{attribute addProperty BoxType "BK1120-0000-0000"}
{attribute addProperty Id "Term_374_KL1002KL1002_D229A9CA00"}
{attribute addProperty CRC "2703046566"}
{attribute addProperty SizeInBites "0"}
{attribute addProperty SizeInBytes "0"}
TYPE A_0001_BK1120_0000_0000_A11D37A6 EXTENDS BK1120_D3F02A0D :
STRUCT
	{attribute addProperty Name "Term_374_KL1002"}
	Term_374_KL1002 : KL1002_D229A9CA;
END_STRUCT
END_TYPE

(* stored: Version 1.2.0.0, ProductVersion 3.1.4024.9
   DUT A_0001_BK1120_0000_0000_A11D37A6: Id {b473f428-9de9-45e7-a080-14dc7feeab8f} *)
